Universal Robots PolyScope program: yj221123.urp

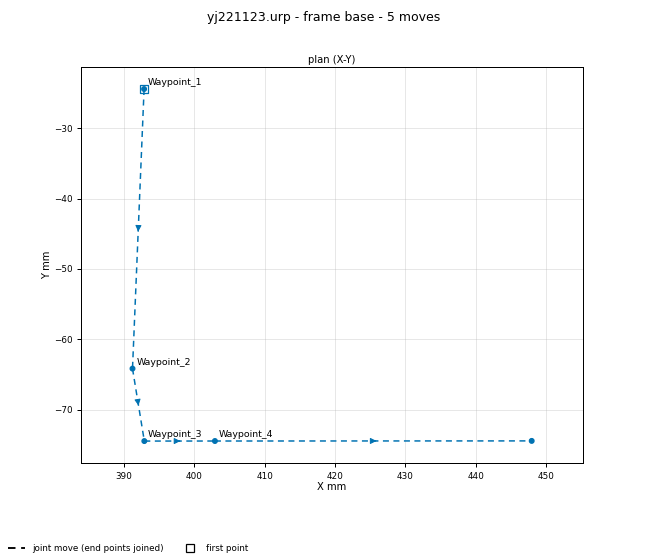
[picture p0: tool path of yj221123.urp in frame base, 5 of 5 moves have a stored position in this frame; points joined in program order, loops and branches not executed]
Program yj221123 (installation=default directory=/programs createdIn=5.11.9.1010452 lastSavedIn=5.11.9.1010452 robotSerialNumber=20225200364)
Calibrated DH parameters: a=[0.00002, -0.569483, -0.54992, -0.00001, -0.000036, 0]; d=[0.180894, -146.691669, 192.918669, -46.053088, 0.119778, 0.115602]; alpha=[1.571425, -0.001534, 0.003359, 1.568739, -1.571477, 0]; deltaTheta=[0, 0.376258, -0.101074, -0.275185, -0.000002, 0]
Robot Program (runOnlyOnce=true)
  MoveJ speed 10 deg/s, acceleration 80 deg/s^2 (useActiveTCP=true) feature=Base
    Waypoint Waypoint_1: motionParameters(blendRadius=0); TCP in base x=392.866 y=-24.44 z=31.99 mm, rx=-3.1416 ry=0.0001 rz=0.0001 rad; joints [22.67, -59.786, -138.912, 288.734, 90.229, -67.382] deg; TCP offset x=0 y=0 z=380 mm, rx=0 ry=0 rz=0 rad
    Waypoint Waypoint_2: motionParameters(blendRadius=0); TCP in base x=391.218 y=-64.177 z=31.997 mm, rx=3.1416 ry=-0.0001 rz=-0.0001 rad; joints [16.717, -60.207, -138.729, 288.971, 90.225, -73.331] deg; TCP offset x=0 y=0 z=380 mm, rx=0 ry=0 rz=0 rad
    Waypoint Waypoint_3: motionParameters(jointSpeed=1.047198 jointAcceleration=1.396263 cartesianSpeed=0.25 cartesianAcceleration=1.2 blendRadius=0.01); TCP in base x=392.898 y=-74.476 z=32.007 mm, rx=2.2214 ry=2.2214 rz=0.0001 rad; joints [15.059, -60.71, -138.507, 289.26, 90.223, -164.992] deg; TCP offset x=0 y=0 z=380 mm, rx=0 ry=0 rz=0 rad
    Waypoint Waypoint_4: motionParameters(blendRadius=0); TCP in base x=402.933 y=-74.468 z=32.033 mm, rx=2.2214 ry=2.2214 rz=0.0002 rad; joints [14.65, -62.152, -137.846, 290.043, 90.224, -165.396] deg; TCP offset x=0 y=0 z=380 mm, rx=0 ry=0 rz=0 rad
    Waypoint Waypoint_5: TCP in base x=447.958 y=-74.452 z=32.067 mm, rx=2.2214 ry=2.2214 rz=0.0003 rad; joints [13.076, -68.249, -134.688, 292.987, 90.217, -166.954] deg; TCP offset x=0 y=0 z=380 mm, rx=0 ry=0 rz=0 rad
